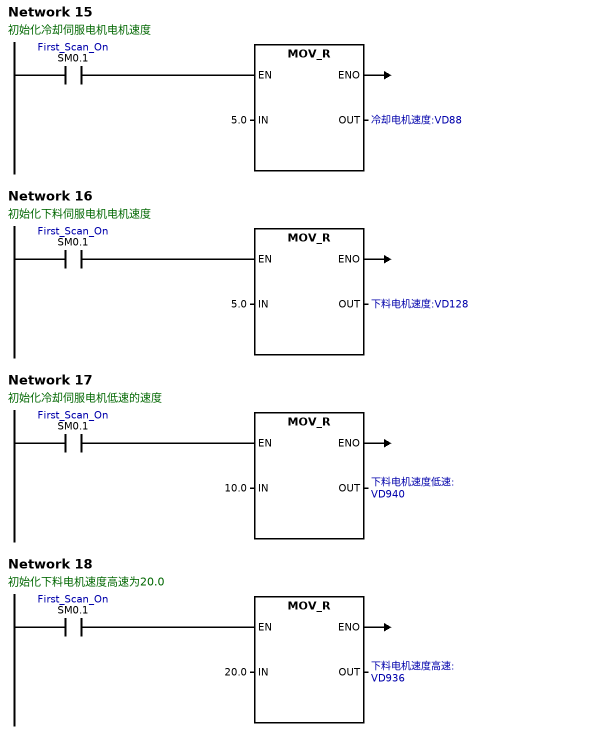
[picture p24: SBR20 networks 15-18]
Network 15
// 初始化冷却伺服电机电机速度
LD     First_Scan_On:SM0.1
MOVR   5.0, 冷却电机速度:VD88
Network 16
// 初始化下料伺服电机电机速度
LD     First_Scan_On:SM0.1
MOVR   5.0, 下料电机速度:VD128
Network 17
// 初始化冷却伺服电机低速的速度
LD     First_Scan_On:SM0.1
MOVR   10.0, 下料电机速度低速:VD940
Network 18
// 初始化下料电机速度高速为20.0
LD     First_Scan_On:SM0.1
MOVR   20.0, 下料电机速度高速:VD936
END_SUBROUTINE_BLOCK

SUBROUTINE_BLOCK 故障报警:SBR21
TITLE=子程序注释
BEGIN
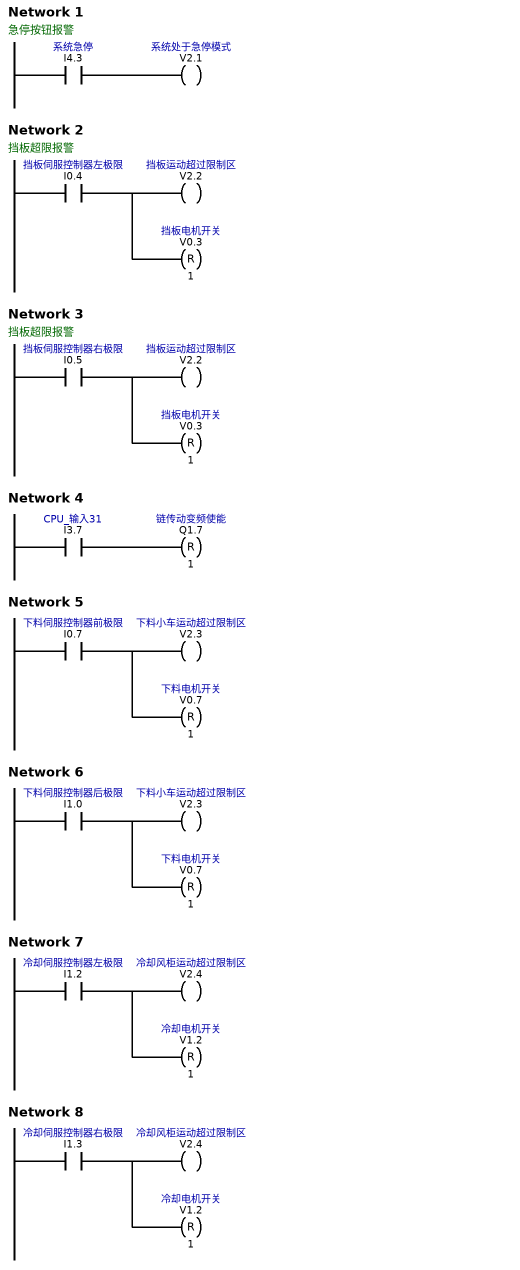
Network 1
// 急停按钮报警
LD     系统急停:I4.3
=      系统处于急停模式:V2.1
Network 2
// 挡板超限报警
LD     挡板伺服控制器左极限:I0.4
=      挡板运动超过限制区:V2.2
R      挡板电机开关:V0.3, 1
Network 3
// 挡板超限报警
LD     挡板伺服控制器右极限:I0.5
=      挡板运动超过限制区:V2.2
R      挡板电机开关:V0.3, 1
Network 4
LD     CPU_输入31:I3.7
R      链传动变频使能:Q1.7, 1
Network 5
LD     下料伺服控制器前极限:I0.7
=      下料小车运动超过限制区:V2.3
R      下料电机开关:V0.7, 1
Network 6
LD     下料伺服控制器后极限:I1.0
=      下料小车运动超过限制区:V2.3
R      下料电机开关:V0.7, 1
Network 7
LD     冷却伺服控制器左极限:I1.2
=      冷却风柜运动超过限制区:V2.4
R      冷却电机开关:V1.2, 1
Network 8
LD     冷却伺服控制器右极限:I1.3
=      冷却风柜运动超过限制区:V2.4
R      冷却电机开关:V1.2, 1
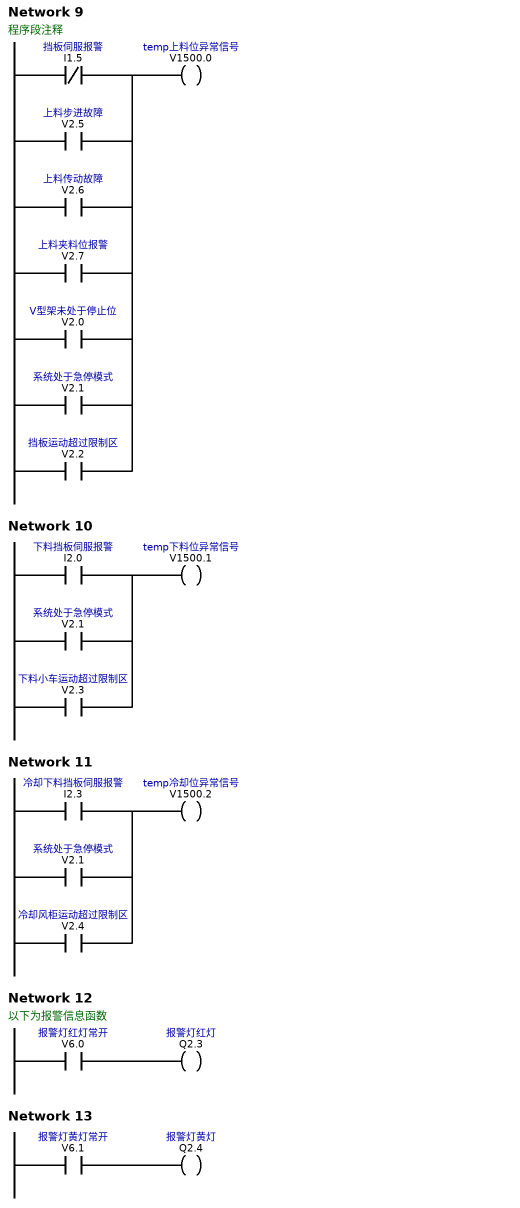
Network 9
// 程序段注释
LDN    挡板伺服报警:I1.5
O      上料步进故障:V2.5
O      上料传动故障:V2.6
O      上料夹料位报警:V2.7
O      V型架未处于停止位:V2.0
O      系统处于急停模式:V2.1
O      挡板运动超过限制区:V2.2
=      temp上料位异常信号:V1500.0
Network 10
LD     下料挡板伺服报警:I2.0
O      系统处于急停模式:V2.1
O      下料小车运动超过限制区:V2.3
=      temp下料位异常信号:V1500.1
Network 11
LD     冷却下料挡板伺服报警:I2.3
O      系统处于急停模式:V2.1
O      冷却风柜运动超过限制区:V2.4
=      temp冷却位异常信号:V1500.2
Network 12
// 以下为报警信息函数
LD     报警灯红灯常开:V6.0
=      报警灯红灯:Q2.3
Network 13
LD     报警灯黄灯常开:V6.1
=      报警灯黄灯:Q2.4
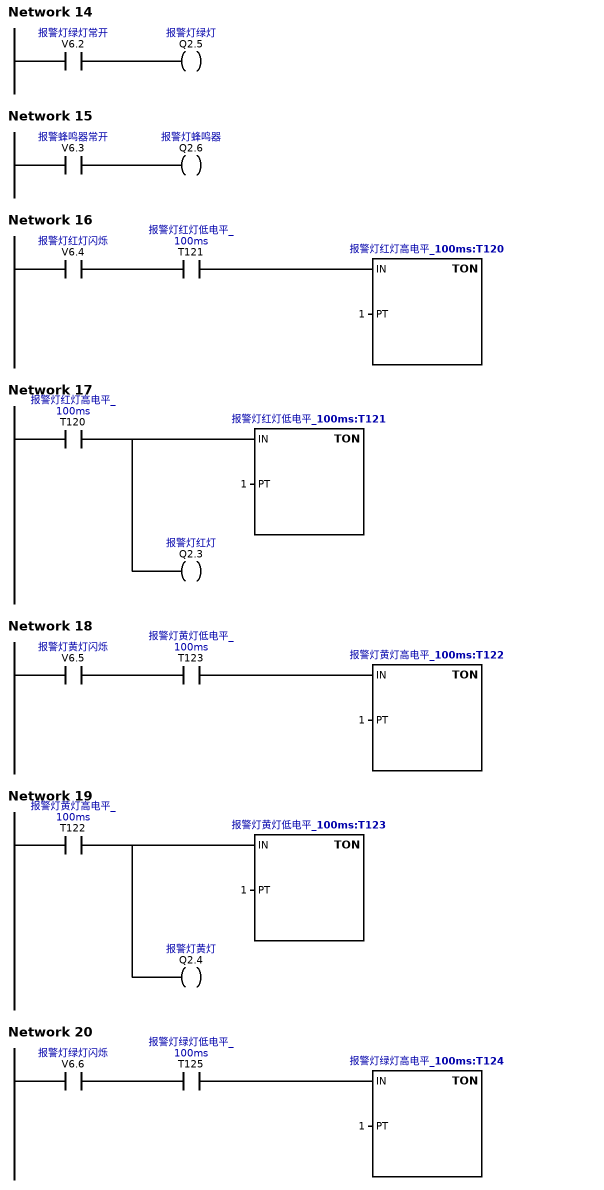
Network 14
LD     报警灯绿灯常开:V6.2
=      报警灯绿灯:Q2.5
Network 15
LD     报警蜂鸣器常开:V6.3
=      报警灯蜂鸣器:Q2.6
Network 16
LD     报警灯红灯闪烁:V6.4
A      报警灯红灯低电平_100ms:T121
TON    报警灯红灯高电平_100ms:T120, 1
Network 17
LD     报警灯红灯高电平_100ms:T120
TON    报警灯红灯低电平_100ms:T121, 1
=      报警灯红灯:Q2.3
Network 18
LD     报警灯黄灯闪烁:V6.5
A      报警灯黄灯低电平_100ms:T123
TON    报警灯黄灯高电平_100ms:T122, 1
Network 19
LD     报警灯黄灯高电平_100ms:T122
TON    报警灯黄灯低电平_100ms:T123, 1
=      报警灯黄灯:Q2.4
Network 20
LD     报警灯绿灯闪烁:V6.6
A      报警灯绿灯低电平_100ms:T125
TON    报警灯绿灯高电平_100ms:T124, 1
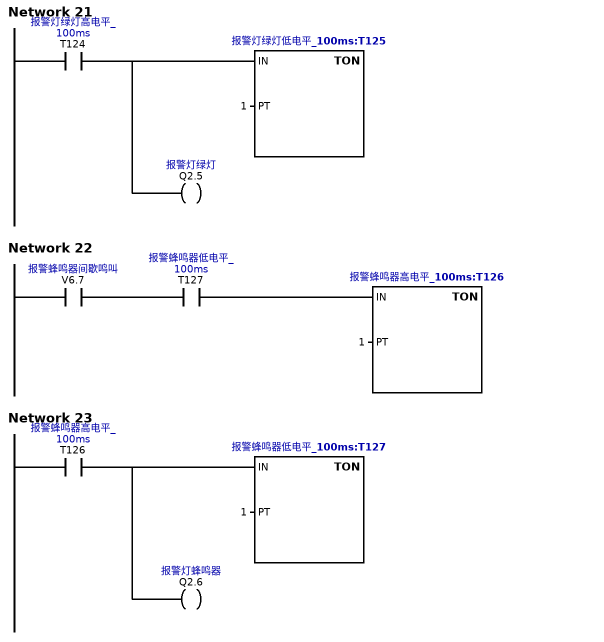
Network 21
LD     报警灯绿灯高电平_100ms:T124
TON    报警灯绿灯低电平_100ms:T125, 1
=      报警灯绿灯:Q2.5
Network 22
LD     报警蜂鸣器间歇鸣叫:V6.7
A      报警蜂鸣器低电平_100ms:T127
TON    报警蜂鸣器高电平_100ms:T126, 1
Network 23
LD     报警蜂鸣器高电平_100ms:T126
TON    报警蜂鸣器低电平_100ms:T127, 1
=      报警灯蜂鸣器:Q2.6
END_SUBROUTINE_BLOCK
